(* LS Electric XG5000 project: XMC_AxisGroup_FBs *)
(* sample programs for axis group function blocks. *)
(* PLC LSPLC *)
(* module base 0 slot 0: Input/Output Module:XMC-DN24 (DC 24V Input 8Points/TR output 16Points) *)
(* module base 0 slot 1: Internal Analog Input/Output:XMF-AH04E (A/D voltage/current 2 channels, D/A voltage 2 channels) *)
(* task Periodic Task: Kind=2 *)
(* task Initialization Task: Kind=1 *)
(* task NC Program: Kind=6 *)

PROGRAM ECAT_Connect_Example (* task: Scan Program *)
VAR
    Connect_Error : BOOL; (* status that LS_Connect has an error *)
    Connect_ErrorID : WORD; (* LS_Connect Error number *)
    Connect_INST : LS_CONNECT; (* LS_Connect fb *)
    Disconnect_Error : BOOL; (* status that LS_Disconnect has an error *)
    Disconnect_ErrorID : WORD; (* Error Number for LS_Disconnect FB *)
    Disconnect_INST : LS_DISCONNECT; (* LS_Disconnect fb *)
    Execute_Connect : BOOL; (* Execute LS_Connect fb *)
    Execute_Disconnect : BOOL; (* execute LS_Disconnect fb *)
END_VAR

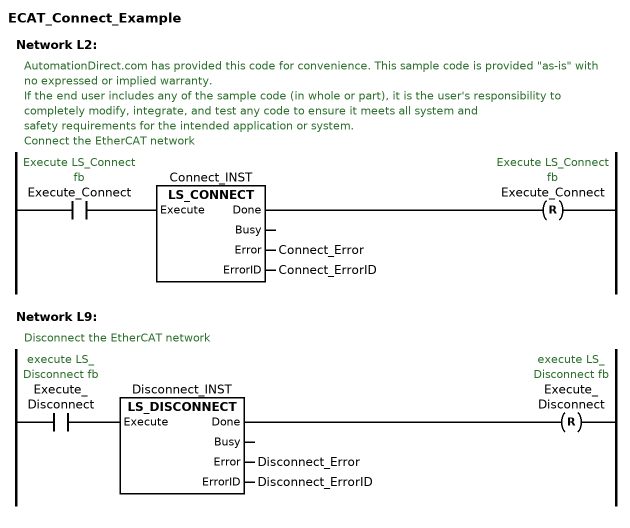
(* AutomationDirect.com has provided this code for convenience. This sample code is provided "as-is" with no expressed or implied warranty. / If the end user includes any of the sample code (in whole or part), it is the user's responsibility to completely modify, integrate, and test any code to ensure it meets all system and / safety requirements for the intended application or system. *)
(* Connect the EtherCAT network *)
(* Rung L2 *)
Connect_INST(Execute := Execute_Connect, Error => Connect_Error, ErrorID => Connect_ErrorID);
IF Connect_INST.Done THEN Execute_Connect := FALSE; END_IF;
(* Disconnect the EtherCAT network *)
(* Rung L9 *)
Disconnect_INST(Execute := Execute_Disconnect, Error => Disconnect_Error, ErrorID => Disconnect_ErrorID);
IF Disconnect_INST.Done THEN Execute_Disconnect := FALSE; END_IF;
END_PROGRAM

PROGRAM MC_AddAxisToGroup_Example (* task: Scan Program *)
(* Example of MC_AddAxisToGroup function block *)
VAR
    AddToGroup_AxesGroup : UINT; (* group to add axis too *)
    AddToGroup_Axis : UINT; (* axis to add to the group *)
    AddToGroup_Busy : BOOL; (* busy status for MC_AddAxisToGroup *)
    AddToGroup_Error : BOOL; (* error status for MC_AddAxisToGroup *)
    AddToGroup_ErrorID : WORD; (* error identification for MC_AddAxisToGroup fb *)
    AddToGroup_IdentInGroup : UINT; (* ID number for the axis *)
    AddToGroup_INST : MC_ADDAXISTOGROUP; (* MC_AddAxisToGroup function block *)
    All_Axes_Ready : BOOL; (* flag that all axes are ready *)
    Execute_AddToGroup : BOOL; (* execute MC_AddAxisToGroup function block *)
END_VAR

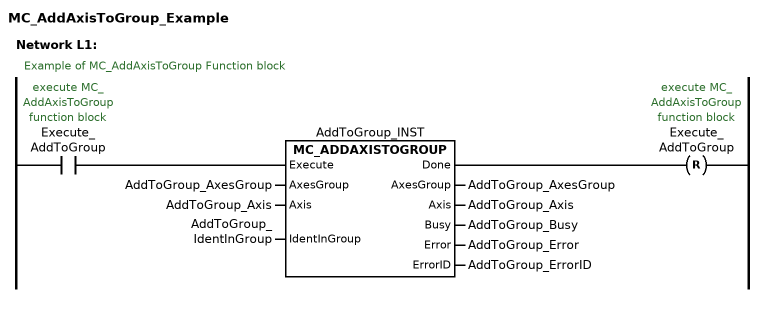
(* Example of MC_AddAxisToGroup Function block *)
(* Rung L1 *)
AddToGroup_INST(Execute := Execute_AddToGroup, AxesGroup := AddToGroup_AxesGroup, Axis := AddToGroup_Axis, IdentInGroup := AddToGroup_IdentInGroup, AxesGroup => AddToGroup_AxesGroup, Axis => AddToGroup_Axis, Busy => AddToGroup_Busy, Error => AddToGroup_Error, ErrorID => AddToGroup_ErrorID);
IF AddToGroup_INST.Done THEN Execute_AddToGroup := FALSE; END_IF;
END_PROGRAM

PROGRAM MC_RemoveAxisFromGroup (* task: Scan Program *)
(* example program for MC_RemoveAxisFromGroup function block *)
VAR
    Execute_RemoveFromGroup : BOOL; (* command to execute MC_RemoveAxisFromGroup fb *)
    GroupRemove_AxesGroup : UINT; (* Group number to remove axis from *)
    GroupRemove_Busy : BOOL; (* busy status *)
    GroupRemove_Error : BOOL; (* error status of MC_RemoveAxisFromGroup *)
    GroupRemove_ErrorID : WORD; (* Error identification for MC_RemoveAxisFromGroup *)
    GroupRemove_IdentInGroup : UINT; (* Identification number of axis to remove *)
    RemoveFromGroup_INST : MC_REMOVEAXISFROMGROUP; (* MC_RemoveAxisFromGroup function block *)
END_VAR

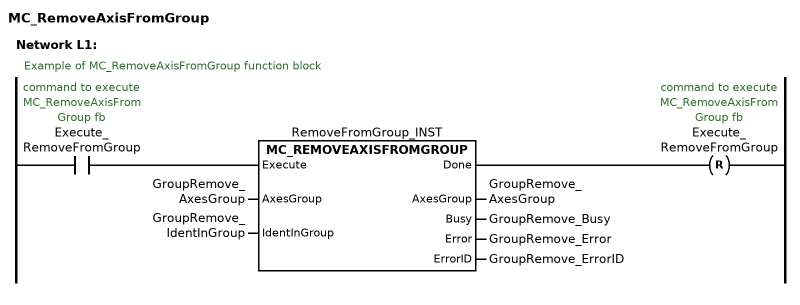
(* Example of MC_RemoveAxisFromGroup function block *)
(* Rung L1 *)
RemoveFromGroup_INST(Execute := Execute_RemoveFromGroup, AxesGroup := GroupRemove_AxesGroup, IdentInGroup := GroupRemove_IdentInGroup, AxesGroup => GroupRemove_AxesGroup, Busy => GroupRemove_Busy, Error => GroupRemove_Error, ErrorID => GroupRemove_ErrorID);
IF RemoveFromGroup_INST.Done THEN Execute_RemoveFromGroup := FALSE; END_IF;
END_PROGRAM

PROGRAM MC_UngroupAllAxes_Example (* task: Scan Program *)
(* program example for MC_UngroupAllAxes function block *)
VAR
    Execute_UngroupAll : BOOL; (* execute MC_UngroupAllAxes function block *)
    UngroupAll_AxesGroup : UINT; (* group number to remove all axes from *)
    UngroupAll_Busy : BOOL; (* busy status for MC_UngroupAllAxes *)
    UngroupAll_Error : BOOL; (* error status for MC_UngroupAllAxes *)
    UngroupAll_ErrorID : WORD; (* error identification for MC_UngroupAllAxes *)
    UngroupAll_INST : MC_UNGROUPALLAXES; (* MC_UngroupAllAxes function block *)
END_VAR

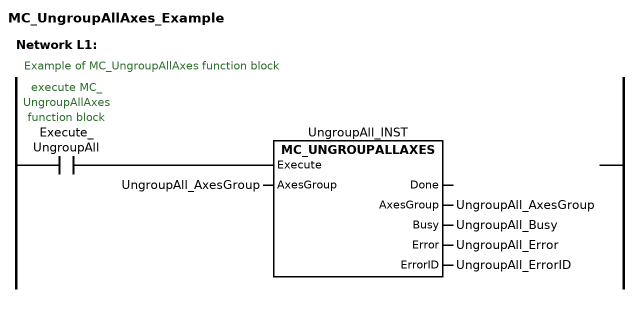
(* Example of MC_UngroupAllAxes function block *)
(* Rung L1 *)
UngroupAll_INST(Execute := Execute_UngroupAll, AxesGroup := UngroupAll_AxesGroup, AxesGroup => UngroupAll_AxesGroup, Busy => UngroupAll_Busy, Error => UngroupAll_Error, ErrorID => UngroupAll_ErrorID);
END_PROGRAM

PROGRAM MC_GroupEnable_Example (* task: Scan Program *)
(* program example for MC_GroupEnable function block *)
VAR
    Execute_GroupEnable : BOOL; (* execute MC_GroupEnable fb *)
    GroupEnable_AxesGroup : UINT; (* Motion Group to enable *)
    GroupEnable_Busy : BOOL; (* Busy status for MC_GroupEnable *)
    GroupEnable_Error : BOOL; (* Error status for MC_GroupEnable fb *)
    GroupEnable_ErrorID : WORD; (* Error identification for MC_GroupEnable *)
    GroupEnable_INST : MC_GROUPENABLE; (* MC_GroupEnable function block *)
END_VAR

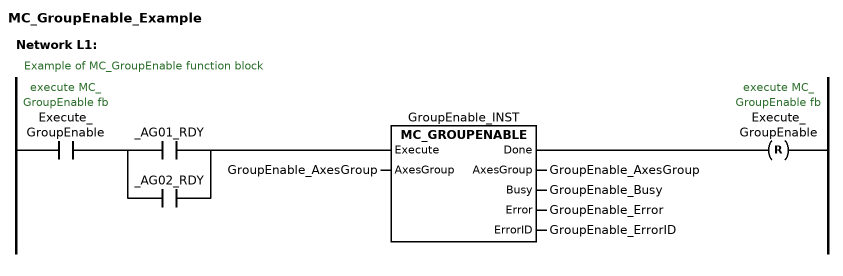
(* Example of MC_GroupEnable function block *)
(* Rung L1 *)
GroupEnable_INST(Execute := Execute_GroupEnable AND (_AG01_RDY OR _AG02_RDY), AxesGroup := GroupEnable_AxesGroup, AxesGroup => GroupEnable_AxesGroup, Busy => GroupEnable_Busy, Error => GroupEnable_Error, ErrorID => GroupEnable_ErrorID);
IF GroupEnable_INST.Done THEN Execute_GroupEnable := FALSE; END_IF;
END_PROGRAM

PROGRAM MC_GroupDisable_Example (* task: Scan Program *)
(* example of of MC_GroupDisable function block *)
VAR
    Execute_GroupDisable : BOOL; (* execute MC_GroupDisable function block *)
    GroupDisable_AxesGroup : UINT; (* Group to disable *)
    GroupDisable_Busy : BOOL; (* busy status for MC_GroupDisable *)
    GroupDisable_Error : BOOL; (* error status for MC_GroupDisable *)
    GroupDisable_ErrorID : WORD; (* error identification for MC_GroupDisable fb *)
    GroupDisable_INST : MC_GROUPDISABLE; (* MC_GroupDisable function block *)
END_VAR

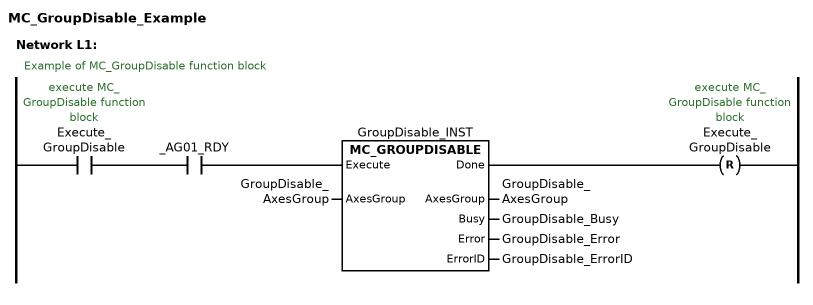
(* Example of MC_GroupDisable function block *)
(* Rung L1 *)
GroupDisable_INST(Execute := Execute_GroupDisable AND _AG01_RDY, AxesGroup := GroupDisable_AxesGroup, AxesGroup => GroupDisable_AxesGroup, Busy => GroupDisable_Busy, Error => GroupDisable_Error, ErrorID => GroupDisable_ErrorID);
IF GroupDisable_INST.Done THEN Execute_GroupDisable := FALSE; END_IF;
END_PROGRAM

PROGRAM MC_GroupPower_Example (* task: Scan Program *)
(* MC_GroupPower function block example program *)
VAR
    Execute_GroupPower : BOOL; (* execute MC_GroupPower function block *)
    GroupPower_AxesGroup : UINT; (* Motion group to power on *)
    GroupPower_Error : BOOL; (* error status of MC_GroupPower function block *)
    GroupPower_ErrorID : WORD; (* error identification for MC_GroupPower *)
    GroupPower_INST : MC_GROUPPOWER; (* MC_GroupPower function block *)
    GroupPower_Status : BOOL; (* MC_GroupPower fb status *)
    GroupPower_Valid : BOOL; (* valid status of MC_GroupPower *)
END_VAR

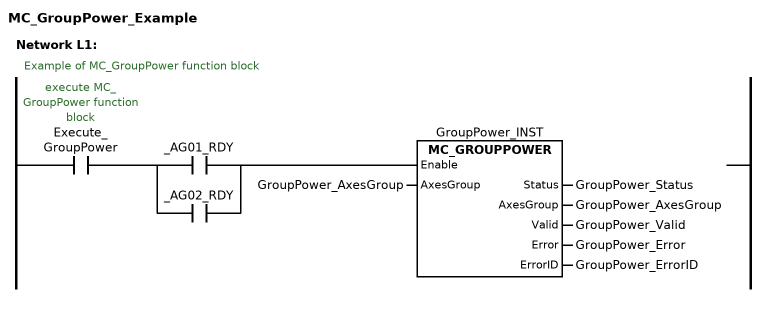
(* Example of MC_GroupPower function block *)
(* Rung L1 *)
GroupPower_INST(Enable := Execute_GroupPower AND (_AG01_RDY OR _AG02_RDY), AxesGroup := GroupPower_AxesGroup, Status => GroupPower_Status, AxesGroup => GroupPower_AxesGroup, Valid => GroupPower_Valid, Error => GroupPower_Error, ErrorID => GroupPower_ErrorID);
END_PROGRAM

PROGRAM MC_GroupHome_Example (* task: Scan Program *)
(* program example for MC_GroupHome function block *)
VAR
    Execute_GroupHome : BOOL; (* Execute MC_GroupHome function block *)
    GroupHome_Aborted : BOOL; (* aborted status for MC_GroupHome *)
    GroupHome_Active : BOOL; (* active status for MC_GroupHome *)
    GroupHome_AxesGroup : UINT; (* Motion group to home *)
    GroupHome_Busy : BOOL; (* busy status for MC_GroupHome *)
    GroupHome_Error : BOOL; (* error status for MC_GroupHome *)
    GroupHome_ErrorID : WORD; (* error identification for MC_GroupHome *)
    GroupHome_INST : MC_GROUPHOME; (* MC_GroupHome function block *)
    GroupHome_Position : ARRAY[0..9] OF LREAL; (* array of positions for MC_GroupHome *)
END_VAR

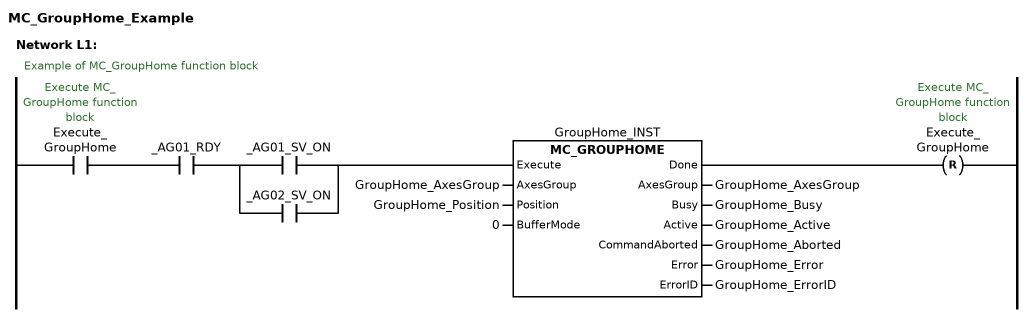
(* Example of MC_GroupHome function block *)
(* Rung L1 *)
GroupHome_INST(Execute := Execute_GroupHome AND _AG01_RDY AND (_AG01_SV_ON OR _AG02_SV_ON), AxesGroup := GroupHome_AxesGroup, Position := GroupHome_Position, BufferMode := 0, AxesGroup => GroupHome_AxesGroup, Busy => GroupHome_Busy, Active => GroupHome_Active, CommandAborted => GroupHome_Aborted, Error => GroupHome_Error, ErrorID => GroupHome_ErrorID);
IF GroupHome_INST.Done THEN Execute_GroupHome := FALSE; END_IF;
END_PROGRAM

PROGRAM MC_GroupSetPosition_Example (* task: Scan Program *)
(* example program for MC_GroupSetPosition and MC_GroupSetPosition2 *)
VAR
    Execute_GroupSetPosition : BOOL; (* execute the MC_GroupSetPosition function block *)
    SetPosition_Aborted : BOOL; (* aborted status for MC_GroupSetPosition *)
    SetPosition_AxesGroup : UINT; (* motion group for MC_GroupSetPosition fb *)
    SetPosition_Busy : BOOL; (* busy status for MC_GroupSetPosition *)
    SetPosition_Error : BOOL; (* error status for MC_GroupSetPosition *)
    SetPosition_ErrorID : WORD; (* error identification for MC_GroupSetPosition *)
    SetPosition_INST : MC_GROUPSETPOSITION; (* MC_GroupSetPosition function block *)
    SetPosition_Position : ARRAY[0..9] OF LREAL; (* positions to set for axes in MC_GroupSetPosition *)
    SetPosition_Relative : BOOL; (* set as relative or absolute position change *)
END_VAR

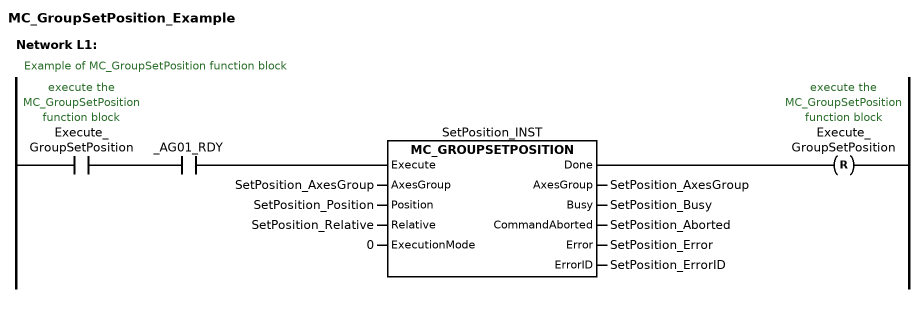
(* Example of MC_GroupSetPosition function block *)
(* Rung L1 *)
SetPosition_INST(Execute := Execute_GroupSetPosition AND _AG01_RDY, AxesGroup := SetPosition_AxesGroup, Position := SetPosition_Position, Relative := SetPosition_Relative, ExecutionMode := 0, AxesGroup => SetPosition_AxesGroup, Busy => SetPosition_Busy, CommandAborted => SetPosition_Aborted, Error => SetPosition_Error, ErrorID => SetPosition_ErrorID);
IF SetPosition_INST.Done THEN Execute_GroupSetPosition := FALSE; END_IF;
END_PROGRAM

PROGRAM MC_GroupStop_Halt_Example (* task: Scan Program *)
(* example program for MC_GroupStop and MC_GroupHalt function blocks *)
VAR
    Execute_GroupHalt : BOOL; (* execute MC_GroupHalt function block *)
    Execute_GroupStop : BOOL; (* execute MC_GroupStop function block *)
    GroupHalt_Aborted : BOOL; (* aborted status of MC_GroupHalt *)
    GroupHalt_Active : BOOL; (* Active status of MC_GroupHalt *)
    GroupHalt_AxesGroup : UINT; (* motion axis group for MC_GroupHalt *)
    GroupHalt_Busy : BOOL; (* busy status of MC_GroupHalt *)
    GroupHalt_Deceleration : LREAL; (* deceleration for MC_GroupHalt *)
    GroupHalt_Error : BOOL; (* error status of MC_GroupHalt *)
    GroupHalt_ErrorID : WORD; (* error identification of MC_GroupHalt *)
    GroupHalt_INST : MC_GROUPHALT; (* MC_GroupHalt function block *)
    GroupHalt_Jerk : LREAL; (* Jerk value for MC_GroupHalt *)
    GroupStop_Aborted : BOOL; (* aborted status for MC_GroupStop *)
    GroupStop_AxesGroup : UINT; (* motion group to stop motion for *)
    GroupStop_Busy : BOOL; (* busy status for MC_GroupSTop *)
    GroupStop_Deceleration : LREAL; (* deceleration for MC_GroupStop fb *)
    GroupStop_Error : BOOL; (* error status for MC_GroupStop *)
    GroupStop_ErrorID : WORD; (* error identification for MC_GroupStop *)
    GroupStop_INST : MC_GROUPSTOP; (* MC_GroupStop function block *)
    GroupStop_Jerk : LREAL; (* Jerk value for MC_GroupStop *)
END_VAR

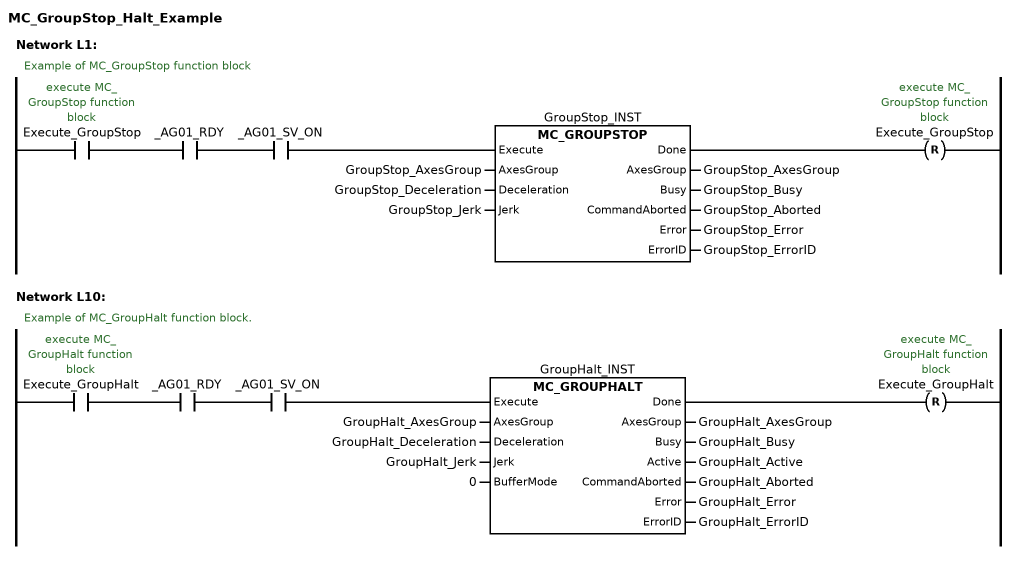
(* Example of MC_GroupStop function block *)
(* Rung L1 *)
GroupStop_INST(Execute := Execute_GroupStop AND _AG01_RDY AND _AG01_SV_ON, AxesGroup := GroupStop_AxesGroup, Deceleration := GroupStop_Deceleration, Jerk := GroupStop_Jerk, AxesGroup => GroupStop_AxesGroup, Busy => GroupStop_Busy, CommandAborted => GroupStop_Aborted, Error => GroupStop_Error, ErrorID => GroupStop_ErrorID);
IF GroupStop_INST.Done THEN Execute_GroupStop := FALSE; END_IF;
(* Example of MC_GroupHalt function block. *)
(* Rung L10 *)
GroupHalt_INST(Execute := Execute_GroupHalt AND _AG01_RDY AND _AG01_SV_ON, AxesGroup := GroupHalt_AxesGroup, Deceleration := GroupHalt_Deceleration, Jerk := GroupHalt_Jerk, BufferMode := 0, AxesGroup => GroupHalt_AxesGroup, Busy => GroupHalt_Busy, Active => GroupHalt_Active, CommandAborted => GroupHalt_Aborted, Error => GroupHalt_Error, ErrorID => GroupHalt_ErrorID);
IF GroupHalt_INST.Done THEN Execute_GroupHalt := FALSE; END_IF;
END_PROGRAM

PROGRAM MC_GroupReset_Example (* task: Scan Program *)
(* example program for MC_GroupReset function block *)
VAR
    Execute_GroupReset : BOOL; (* execute MC_GroupReset function block *)
    GroupReset_AxesGroup : UINT; (* axis group for MC_GroupReset *)
    GroupReset_Busy : BOOL; (* busy status for MC_GroupReset *)
    GroupReset_Error : BOOL; (* error status for MC_GroupStatus *)
    GroupReset_ErrorID : WORD; (* error identification for MC_GroupReset *)
    GroupReset_INST : MC_GROUPRESET; (* MC_GroupReset function block *)
END_VAR

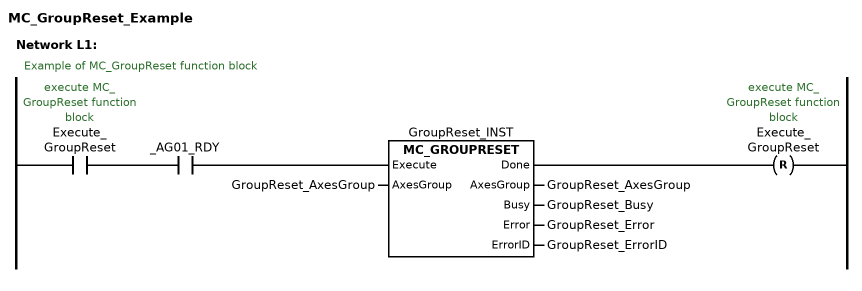
(* Example of MC_GroupReset function block *)
(* Rung L1 *)
GroupReset_INST(Execute := Execute_GroupReset AND _AG01_RDY, AxesGroup := GroupReset_AxesGroup, AxesGroup => GroupReset_AxesGroup, Busy => GroupReset_Busy, Error => GroupReset_Error, ErrorID => GroupReset_ErrorID);
IF GroupReset_INST.Done THEN Execute_GroupReset := FALSE; END_IF;
END_PROGRAM

PROGRAM MC_MoveLinearAbsolute_Example (* task: Scan Program *)
(* example program for MC_MoveLinearAbsolute function block. *)
VAR
    Execute_MoveLinearAbs : BOOL; (* Execute MC_MoveLinearAbsolute function block *)
    MoveLinearAbs_Aborted : BOOL; (* aborted status for MC_MoveLinearAbsolute *)
    MoveLinearAbs_Acceleration : LREAL; (* acceleration for MC_MoveLinearAbsolute *)
    MoveLinearAbs_Active : BOOL; (* active status for MC_MoveLinearAbsolute *)
    MoveLinearAbs_AxesGroup : UINT; (* axis group for MC_MoveLinearAbsolute fb *)
    MoveLinearAbs_Busy : BOOL; (* busy status for MC_MoveLinearAbsolute *)
    MoveLinearAbs_Deceleration : LREAL; (* deceleration for MC_MoveLinearAbsolute *)
    MoveLinearAbs_Error : BOOL; (* error status for MC_MoveLinearAbsolute *)
    MoveLinearAbs_ErrorID : WORD; (* error identification for MC_MoveLinearAbsolute *)
    MoveLinearAbs_INST : MC_MOVELINEARABSOLUTE; (* MC_MoveLinearAbsolute function block *)
    MoveLinearAbs_Jerk : LREAL; (* jerk value for MC_MoveLinearAbsolute *)
    MoveLinearAbs_Position : ARRAY[0..9] OF LREAL; (* position array for MC_MoveLinearAbsolute *)
    MoveLinearAbs_Velocity : LREAL; (* max velocity for MC_MoveLinearAbsolute *)
END_VAR

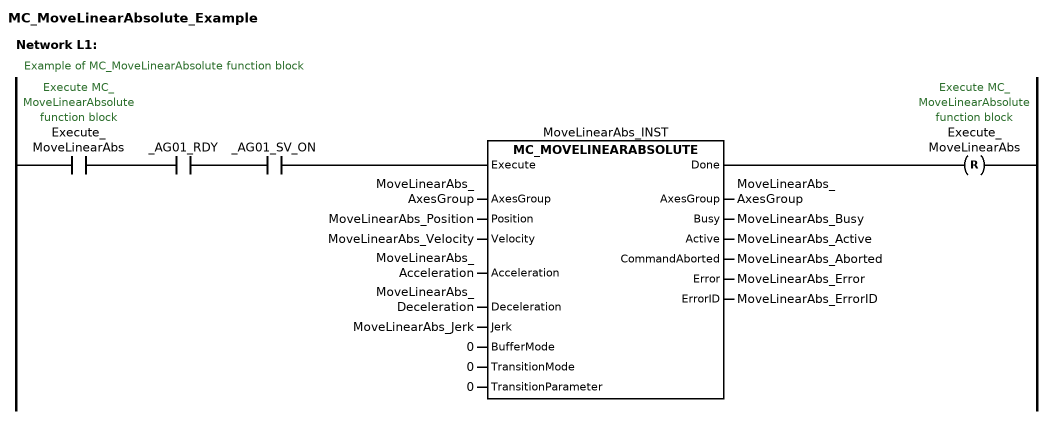
(* Example of MC_MoveLinearAbsolute function block *)
(* Rung L1 *)
MoveLinearAbs_INST(Execute := Execute_MoveLinearAbs AND _AG01_RDY AND _AG01_SV_ON, AxesGroup := MoveLinearAbs_AxesGroup, Position := MoveLinearAbs_Position, Velocity := MoveLinearAbs_Velocity, Acceleration := MoveLinearAbs_Acceleration, Deceleration := MoveLinearAbs_Deceleration, Jerk := MoveLinearAbs_Jerk, BufferMode := 0, TransitionMode := 0, TransitionParameter := 0, AxesGroup => MoveLinearAbs_AxesGroup, Busy => MoveLinearAbs_Busy, Active => MoveLinearAbs_Active, CommandAborted => MoveLinearAbs_Aborted, Error => MoveLinearAbs_Error, ErrorID => MoveLinearAbs_ErrorID);
IF MoveLinearAbs_INST.Done THEN Execute_MoveLinearAbs := FALSE; END_IF;
END_PROGRAM

PROGRAM MC_MoveLinearRelative_Example (* task: Scan Program *)
(* example program of MC_MoveLinearRelative function block *)
VAR
    Execute_MoveLinearRelative : BOOL; (* execute MC_MoveLinearRelative function block *)
    MoveLinearRelative_Aborted : BOOL; (* aborted status for MC_MoveLinearRelative *)
    MoveLinearRelative_Acceleration : LREAL; (* acceleration of linear move *)
    MoveLinearRelative_Active : BOOL; (* active status for MC_MoveLinearRelative *)
    MoveLinearRelative_AxesGroup : UINT; (* axis group for MC_MoveLinearRelative *)
    MoveLinearRelative_Busy : BOOL; (* busy status for MC_MoveLinearRelative *)
    MoveLinearRelative_Deceleration : LREAL; (* deceleration of linear move *)
    MoveLinearRelative_Distance : ARRAY[0..9] OF LREAL; (* distances for MC_MoveLinearRelative *)
    MoveLinearRelative_Error : BOOL; (* error status for MC_MoveLinearRelative *)
    MoveLinearRelative_ErrorID : WORD; (* error identification for MC_MoveLinearRelative *)
    MoveLinearRelative_INST : MC_MOVELINEARRELATIVE; (* MC_MoveLinearRelative function block *)
    MoveLinearRelative_Jerk : LREAL; (* jerk value for linear move *)
    MoveLinearRelative_Velocity : LREAL; (* velocity of relative move *)
END_VAR

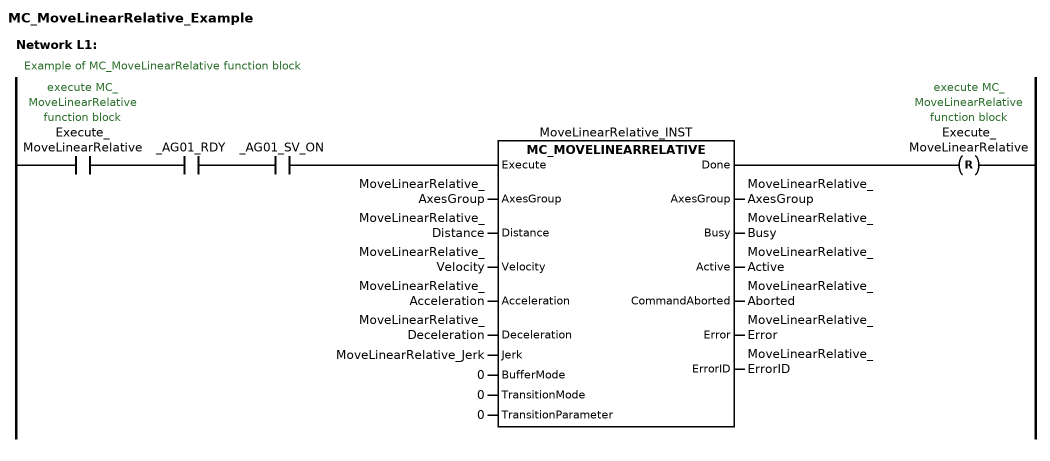
(* Example of MC_MoveLinearRelative function block *)
(* Rung L1 *)
MoveLinearRelative_INST(Execute := Execute_MoveLinearRelative AND _AG01_RDY AND _AG01_SV_ON, AxesGroup := MoveLinearRelative_AxesGroup, Distance := MoveLinearRelative_Distance, Velocity := MoveLinearRelative_Velocity, Acceleration := MoveLinearRelative_Acceleration, Deceleration := MoveLinearRelative_Deceleration, Jerk := MoveLinearRelative_Jerk, BufferMode := 0, TransitionMode := 0, TransitionParameter := 0, AxesGroup => MoveLinearRelative_AxesGroup, Busy => MoveLinearRelative_Busy, Active => MoveLinearRelative_Active, CommandAborted => MoveLinearRelative_Aborted, Error => MoveLinearRelative_Error, ErrorID => MoveLinearRelative_ErrorID);
IF MoveLinearRelative_INST.Done THEN Execute_MoveLinearRelative := FALSE; END_IF;
END_PROGRAM

PROGRAM MC_MoveCircularAbsolute_Example (* task: Scan Program *)
(* example of MC_MoveCircularAbsolute function block *)
VAR
    Execute_MoveCircularAbs : BOOL; (* execute MC_MoveCircularAbsolute *)
    MoveCircularAbs_Aborted : BOOL; (* aborted status for MC_MoveCircularAbsolute *)
    MoveCircularAbs_Acceleration : LREAL; (* maximum acceleration for MC_MoveCircularAbsolute *)
    MoveCircularAbs_Active : BOOL; (* active status for MC_MoveCircularAbsolute *)
    MoveCircularAbs_AuxPoint : ARRAY[0..2] OF LREAL; (* Auxiliary point for MC_MoveCircularAbsolute *)
    MoveCircularAbs_AxesGroup : UINT; (* axis group for MC_MoveCircularAbsolute *)
    MoveCircularAbs_Busy : BOOL; (* busy status for MC_MoveCircularAbsolute *)
    MoveCircularAbs_CircMode : UINT; (* Circular Mode for MC_MoveCircularAbsolute *)
    MoveCircularAbs_Deceleration : LREAL; (* maximum decleration of MC_MoveCircularAbsolute *)
    MoveCircularAbs_EndPoint : ARRAY[0..2] OF LREAL; (* End point of MC_MoveCircularAbsolute *)
    MoveCircularAbs_Error : BOOL; (* error status for MC_MoveCircularAbsolute *)
    MoveCircularAbs_ErrorID : WORD; (* error identification for MC_MoveCircularAbsolute *)
    MoveCircularAbs_INST : MC_MOVECIRCULARABSOLUTE; (* MC_MoveCircularAbsolute function block *)
    MoveCircularAbs_Jerk : LREAL; (* jerk value of MC_MoveCircularAbsolute *)
    MoveCircularAbs_PathChoice : UINT; (* path choice for MC_MoveCircularAbsolute *)
    MoveCircularAbs_Velocity : LREAL; (* maximum velocity for MC_MoveCircularAbsolute *)
END_VAR

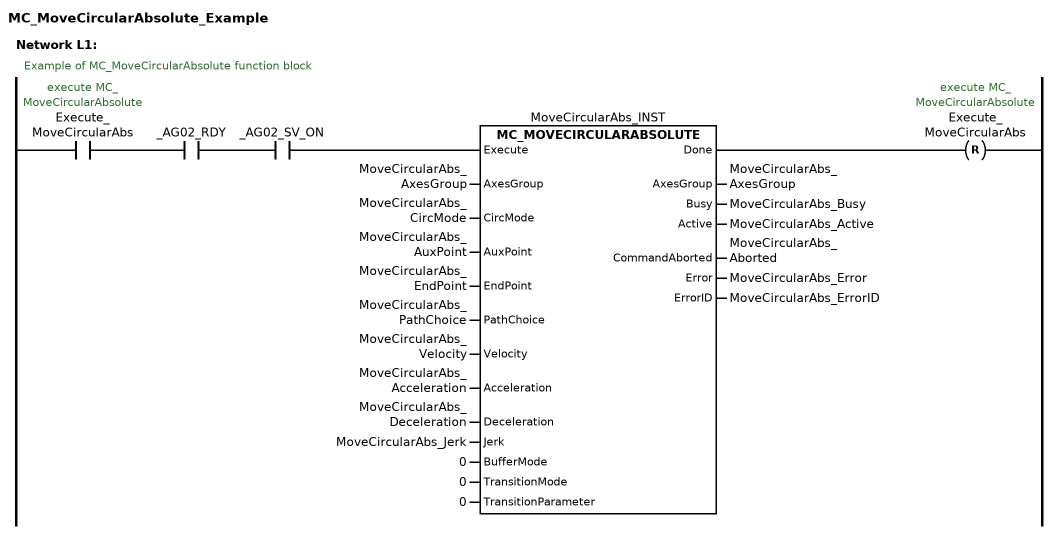
(* Example of MC_MoveCircularAbsolute function block *)
(* Rung L1 *)
MoveCircularAbs_INST(Execute := Execute_MoveCircularAbs AND _AG02_RDY AND _AG02_SV_ON, AxesGroup := MoveCircularAbs_AxesGroup, CircMode := MoveCircularAbs_CircMode, AuxPoint := MoveCircularAbs_AuxPoint, EndPoint := MoveCircularAbs_EndPoint, PathChoice := MoveCircularAbs_PathChoice, Velocity := MoveCircularAbs_Velocity, Acceleration := MoveCircularAbs_Acceleration, Deceleration := MoveCircularAbs_Deceleration, Jerk := MoveCircularAbs_Jerk, BufferMode := 0, TransitionMode := 0, TransitionParameter := 0, AxesGroup => MoveCircularAbs_AxesGroup, Busy => MoveCircularAbs_Busy, Active => MoveCircularAbs_Active, CommandAborted => MoveCircularAbs_Aborted, Error => MoveCircularAbs_Error, ErrorID => MoveCircularAbs_ErrorID);
IF MoveCircularAbs_INST.Done THEN Execute_MoveCircularAbs := FALSE; END_IF;
END_PROGRAM

PROGRAM MC_MoveCircularRelative_Example (* task: Scan Program *)
(* example program for MC_MoveCircularRelative function block *)
VAR
    Execute_MoveCircularRel : BOOL; (* execute MC_MoveCircularRelative function block *)
    MoveCircularRel_Aborted : BOOL; (* aborted status of MC_MoveCircularRelative *)
    MoveCircularRel_Acceleration : LREAL; (* accleration of MC_MoveCircularRelative *)
    MoveCircularRel_Active : BOOL; (* active status for MC_MoveCircularRelative *)
    MoveCircularRel_AuxPoint : ARRAY[0..2] OF LREAL; (* auxiliary point for MC_MoveCircularRelative *)
    MoveCircularRel_AxesGroup : UINT; (* axis group for MC_MoveCircularRelative *)
    MoveCircularRel_Busy : BOOL; (* busy status for MC_MoveCircularRelative *)
    MoveCircularRel_CircMode : UINT; (* circular interpolation mode *)
    MoveCircularRel_Deceleration : LREAL; (* deceleration of MC_MoveCircularRelative *)
    MoveCircularRel_EndPoint : ARRAY[0..2] OF LREAL; (* end point of MC_MoveCircularRelative *)
    MoveCircularRel_Error : BOOL; (* error status of MC_MoveCircularRelative *)
    MoveCircularRel_ErrorID : WORD; (* error identification of MC_MoveCircularRelative *)
    MoveCircularRel_INST : MC_MOVECIRCULARRELATIVE; (* MC_MoveCircularRelative function block *)
    MoveCircularRel_Jerk : LREAL; (* jerk value of MC_MoveCircularRelative *)
    MoveCircularRel_PathChoice : UINT; (* movement direction of MC_MoveCircularRelative *)
    MoveCircularRel_Velocity : LREAL; (* maximum velocity of MC_MoveCircularRelative *)
END_VAR

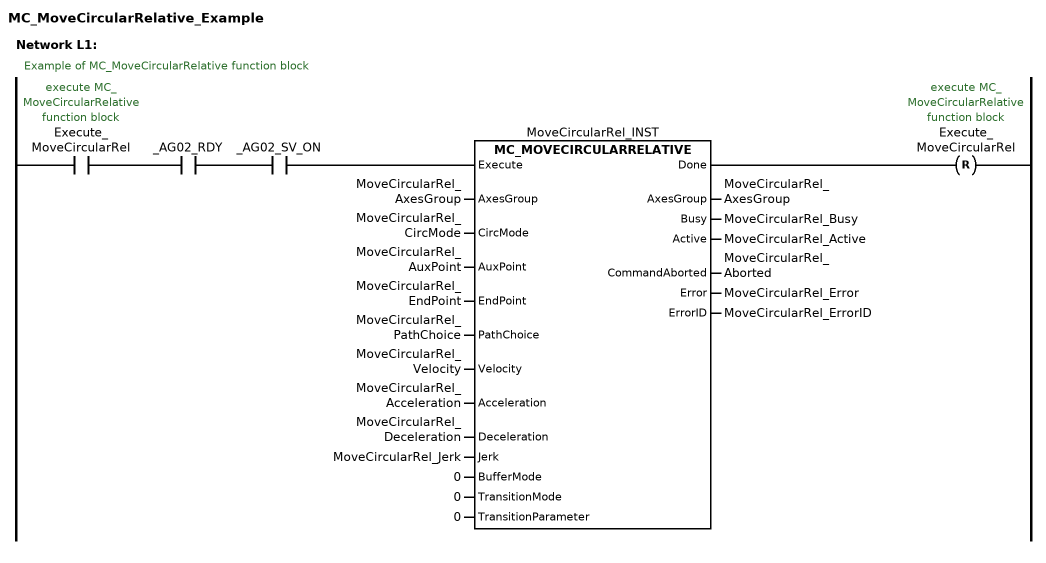
(* Example of MC_MoveCircularRelative function block *)
(* Rung L1 *)
MoveCircularRel_INST(Execute := Execute_MoveCircularRel AND _AG02_RDY AND _AG02_SV_ON, AxesGroup := MoveCircularRel_AxesGroup, CircMode := MoveCircularRel_CircMode, AuxPoint := MoveCircularRel_AuxPoint, EndPoint := MoveCircularRel_EndPoint, PathChoice := MoveCircularRel_PathChoice, Velocity := MoveCircularRel_Velocity, Acceleration := MoveCircularRel_Acceleration, Deceleration := MoveCircularRel_Deceleration, Jerk := MoveCircularRel_Jerk, BufferMode := 0, TransitionMode := 0, TransitionParameter := 0, AxesGroup => MoveCircularRel_AxesGroup, Busy => MoveCircularRel_Busy, Active => MoveCircularRel_Active, CommandAborted => MoveCircularRel_Aborted, Error => MoveCircularRel_Error, ErrorID => MoveCircularRel_ErrorID);
IF MoveCircularRel_INST.Done THEN Execute_MoveCircularRel := FALSE; END_IF;
END_PROGRAM

PROGRAM LS_ReadParameterGroup_Example (* task: Scan Program *)
(* example program for LS_ReadParameterGroup function block *)
VAR
    Execute_ReadParameter : BOOL; (* Execute LS_ReadParameterGroup *)
    ParameterNumber : INT; (* parameter number for LS_ReadGroupParameter *)
    ReadParameter_AxesGroup : UINT; (* axis group for LS_ReadGroupParameter *)
    ReadParameter_Busy : BOOL; (* busy status for LS_ReadGroupParameter *)
    ReadParameter_Error : BOOL; (* error status for LS_ReadGroupParameter *)
    ReadParameter_ErrorID : WORD; (* error identification for LS_ReadGroupParameter *)
    ReadParameter_INST : LS_READGROUPPARAMETER; (* LS_ReadGroupParameter function block *)
    ReadParameter_Valid : BOOL; (* valid status for LS_ReadGroupParameter *)
    ReadParameter_Value : LREAL; (* value of the parameter selected *)
END_VAR

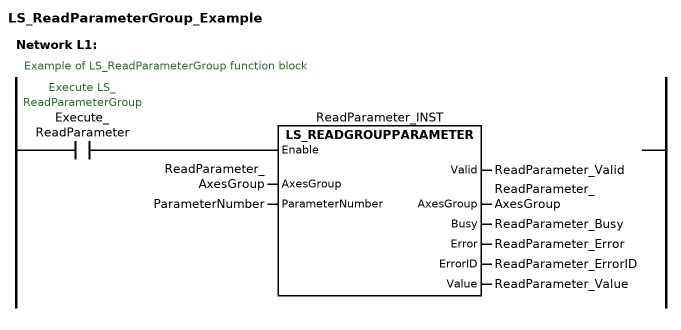
(* Example of LS_ReadParameterGroup function block *)
(* Rung L1 *)
ReadParameter_INST(Enable := Execute_ReadParameter, AxesGroup := ReadParameter_AxesGroup, ParameterNumber := ParameterNumber, Valid => ReadParameter_Valid, AxesGroup => ReadParameter_AxesGroup, Busy => ReadParameter_Busy, Error => ReadParameter_Error, ErrorID => ReadParameter_ErrorID, Value => ReadParameter_Value);
END_PROGRAM

PROGRAM LS_WriteGroupParameter_Example (* task: Scan Program *)
(* example program for LS_WriteGroupParameter *)
VAR
    Execute_WriteParameter : BOOL; (* Execute LS_WriteGroupParameter function block *)
    ParameterNumber : INT; (* parameter number for LS_WriteGroupParameter *)
    WriteParameter_AxesGroup : UINT; (* axis group for LS_WriteGroupParameter *)
    WriteParameter_Busy : BOOL; (* busy status for LS_WriteGroupParameter *)
    WriteParameter_Error : BOOL; (* Error status for LS_WriteGroupParameter *)
    WriteParameter_ErrorID : WORD; (* error identification for LS_WriteGroupParameter *)
    WriteParameter_INST : LS_WRITEGROUPPARAMETER; (* LS_WriteGroupParameter function block *)
    WriteParameter_Value : LREAL; (* value for LS_WriteGroupParameter *)
END_VAR

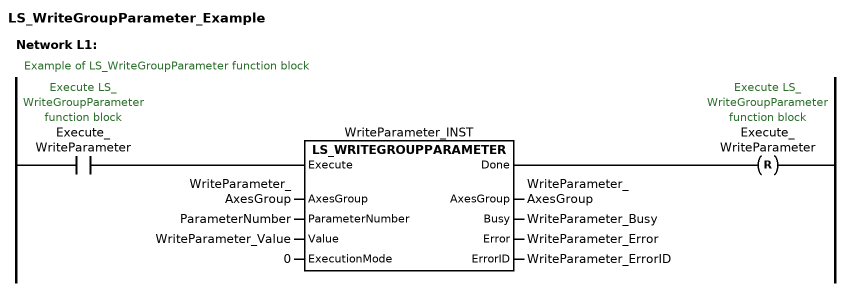
(* Example of LS_WriteGroupParameter function block *)
(* Rung L1 *)
WriteParameter_INST(Execute := Execute_WriteParameter, AxesGroup := WriteParameter_AxesGroup, ParameterNumber := ParameterNumber, Value := WriteParameter_Value, ExecutionMode := 0, AxesGroup => WriteParameter_AxesGroup, Busy => WriteParameter_Busy, Error => WriteParameter_Error, ErrorID => WriteParameter_ErrorID);
IF WriteParameter_INST.Done THEN Execute_WriteParameter := FALSE; END_IF;
END_PROGRAM

PROGRAM MC_GroupSetOverride_Example (* task: Scan Program *)
(* Example program for MC_GroupSetOverride function block *)
VAR
    AxesGroup : UINT; (* Axis group for MC_GroupSetOverride example *)
    LinearRelative_Active : BOOL; (* Active Status for MC_MoveLinearRelative *)
    LinearRelative_Distance : ARRAY[0..9] OF LREAL; (* distance values for MC_MoveLinearRelative *)
    LinearRelative_Error : BOOL; (* error Status for MC_MoveLinearRelative *)
    LinearRelative_ErrorID : WORD; (* error identification for MC_MoveLinearRelative *)
    LinearRelative_INST : MC_MOVELINEARRELATIVE; (* MC_MoveLinearRelative function block *)
    Run_Example : BOOL; (* run the MC_GroupSetOverride example *)
    SetOverride_AccFactor : LREAL; (* acceleration override factor *)
    SetOverride_Busy : BOOL; (* busy status of MC_GroupSetOverride *)
    SetOverride_Enabled : BOOL; (* enabled status for MC_GroupSetOverride *)
    SetOverride_Error : BOOL; (* error status of MC_GroupSetOverride *)
    SetOverride_ErrorID : WORD; (* error identification of MC_GroupSetOverride *)
    SetOverride_INST : MC_GROUPSETOVERRIDE; (* MC_GroupSetOverride function block *)
    SetOverride_JerkFactor : LREAL; (* Jerk override factor *)
    SetOverride_VelFactor : LREAL; (* Override velocity factor *)
END_VAR

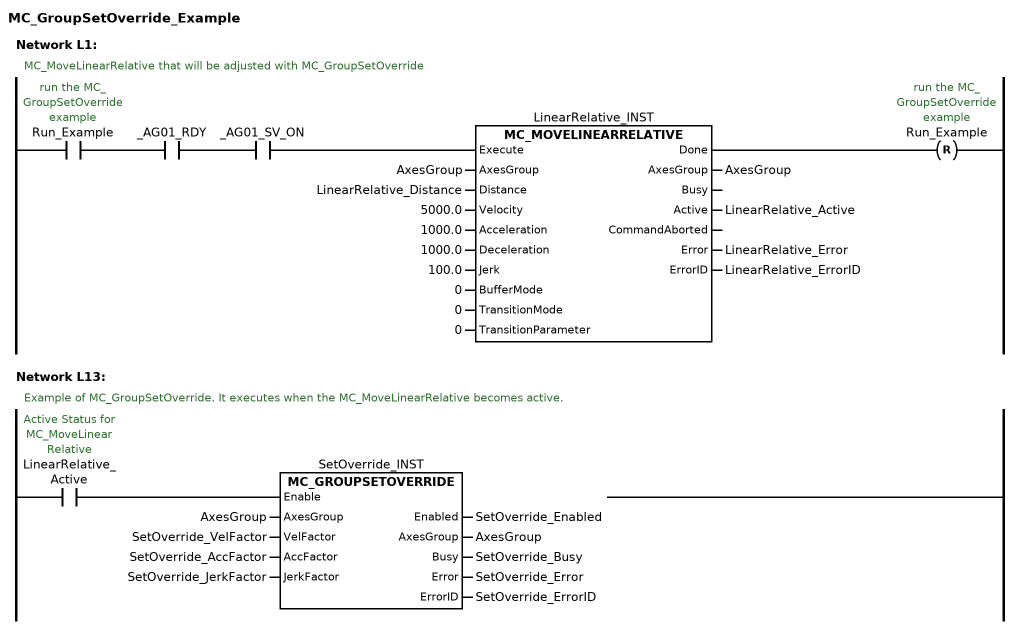
(* MC_MoveLinearRelative that will be adjusted with MC_GroupSetOverride *)
(* Rung L1 *)
LinearRelative_INST(Execute := Run_Example AND _AG01_RDY AND _AG01_SV_ON, AxesGroup := AxesGroup, Distance := LinearRelative_Distance, Velocity := 5000.0, Acceleration := 1000.0, Deceleration := 1000.0, Jerk := 100.0, BufferMode := 0, TransitionMode := 0, TransitionParameter := 0, AxesGroup => AxesGroup, Active => LinearRelative_Active, Error => LinearRelative_Error, ErrorID => LinearRelative_ErrorID);
IF LinearRelative_INST.Done THEN Run_Example := FALSE; END_IF;
(* Example of MC_GroupSetOverride. It executes when the MC_MoveLinearRelative becomes active. *)
(* Rung L13 *)
SetOverride_INST(Enable := LinearRelative_Active, AxesGroup := AxesGroup, VelFactor := SetOverride_VelFactor, AccFactor := SetOverride_AccFactor, JerkFactor := SetOverride_JerkFactor, Enabled => SetOverride_Enabled, AxesGroup => AxesGroup, Busy => SetOverride_Busy, Error => SetOverride_Error, ErrorID => SetOverride_ErrorID);
END_PROGRAM